TYPE ST_LaudaWriteCommands_Temperature :
STRUCT
	TemperatureSet				: STRING := 'OUT_SP_00_';
	ActualExternalTemperature	: STRING := 'OUT_PV_05_';
	OutflowLimmitHigh			: STRING := 'OUT_SP_04_';
	OutflowLimmitLow			: STRING := 'OUT_SP_05_';
	SafetyModeTemperature		: STRING := 'OUT_SP_07_';
END_STRUCT
END_TYPE

(* stored: Version 1.1.0.1, ProductVersion 3.1.4024.12
   DUT ST_LaudaWriteCommands_Temperature: Id {399b56f8-aa49-4ecc-8dca-613452554873} *)
